TYPE ST_SettingsAirTrearment :
STRUCT
	; //To be defined
END_STRUCT
END_TYPE

(* stored: Version 1.1.0.1, ProductVersion 3.1.4024.12
   DUT ST_SettingsAirTrearment: Id {06fc4816-030f-4763-8a01-113573740184} *)
